{attribute 'qualified_only'}
{attribute 'strict'}
{attribute 'to_string'}
TYPE eSkillCommand :
(
	KEINE		:= 0,
	STARTEN		:= 1,
	STOPPEN		:= 2,
	RESETTEN 	:= 3
);
END_TYPE

(* stored: Version 1.1.0.1
   DUT eSkillCommand: Id {1716bd6d-e6b5-4c1d-86bb-a53f9219e577} *)
